Fanuc TP program (LS listing): HOME.ls

/PROG  HOME
/ATTR
OWNER		= MNEDITOR;
COMMENT		= "";
PROG_SIZE	= 150;
CREATE		= DATE 25-07-06  TIME 02:13:40;
MODIFIED	= DATE 25-07-06  TIME 02:14:02;
FILE_NAME	= ;
VERSION		= 0;
LINE_COUNT	= 1;
MEMORY_SIZE	= 518;
PROTECT		= READ_WRITE;
TCD:  STACK_SIZE	= 0,
      TASK_PRIORITY	= 50,
      TIME_SLICE	= 0,
      BUSY_LAMP_OFF	= 0,
      ABORT_REQUEST	= 0,
      PAUSE_REQUEST	= 0;
DEFAULT_GROUP	= 1,*,*,*,*;
CONTROL_CODE	= 00000000 00000000;
/MN
   1:J PR[10:HOME3] 100% FINE    ;
/POS
/END
